TYPE ST_HEATER_STATIC_SETTINGS :
STRUCT
	testTemperature:	REAL := 28.0;
	workTemperature:	REAL := 40.0;
	hysteresis:			REAL := 2.0;
END_STRUCT
END_TYPE

(* stored: Version 1.1.0.1
   DUT ST_HEATER_STATIC_SETTINGS: Id {0b44db92-1a33-4ad1-8bc7-339db9981203} *)
